TYPE ST_RejectReason_PK2_OUT2 :
STRUCT
	Reason	:STRING;
END_STRUCT
END_TYPE

(* stored: Version 1.1.0.1, ProductVersion 3.1.4024.13
   DUT ST_RejectReason_PK2_OUT2: Id {abf24c13-dc63-4fed-b7bc-941e6fa61a23} *)
